// Mitsubishi GX Works2 project: 機電整合丙級第一題-ST   PLC: FX3U/FX3UC

// task Task_01 (event TRUE, interval 0, priority 31): POU_01

PROGRAM POU_01
VAR
  wProgramStep : INT;
  bM17 : BOOL;
  bM24 : BOOL;
  bM44 : BOOL;
  bM122 : BOOL;
  tdT22 : TON;
  bShape : BOOL;
  tdT24 : TON;
  tdT27 : TON;
  tdT29 : TON;
  bPB2 : BOOL;
  tdT123 : TON;
END_VAR
(* 機電整合丙級術科第一題
   Author: Steven Luo
   Date: 2018/09/26
*)

IF M8002 OR NOT X17 THEN (* 開機後或任何狀態按下急停 *)
	wProgramStep := 0;
	ZRST(TRUE, Y0, Y17);
	bM17 := FALSE;
	bM122 := FALSE;
END_IF;

IF NOT X17 THEN (* 按下急停 *)
	RST(TRUE, Y0);
	bM17 := TRUE;
END_IF;

IF X17 AND bM17 THEN (* 放開急停，等待復歸 *)
	wProgramStep := 122;
END_IF;

IF M8002 THEN
	wProgramStep := 21;
END_IF;

IF bM122 THEN
	IF M8013 THEN
		SET(TRUE, Y16); (* 黃燈閃爍 *)
	ELSE
		RST(TRUE, Y16);
	END_IF;
ELSE
	RST(TRUE, Y16);
END_IF;

CASE wProgramStep OF
	21:
		IF X1 AND X4 THEN
			SET(TRUE, Y17); (* 待機，綠燈亮、紅燈滅 *)
			RST(TRUE, Y15);
			RST(TRUE, Y2);
			tdT22(IN := FALSE);
			tdT24(IN := FALSE);
			tdT27(IN := FALSE);
			tdT29(IN := FALSE);
			tdT123(IN := FALSE);
			bM122 := FALSE;
			bM24 := FALSE;
			bM44 := FALSE;
			bPB2 := FALSE;
		END_IF;
		IF X13 AND X17 THEN
			IF X14 THEN (* 指定功能 *)
				RST(TRUE, Y2);
				RST(TRUE, Y4);
				RST(TRUE, Y5);
				IF X7 THEN (* PB1 *)
					SET(TRUE, Y2);
				ELSIF X4 AND X10 THEN (* PB2 *)
					IF X0 THEN
						RST(TRUE, Y0);
					ELSE
						SET(TRUE, Y0);
					END_IF;
				ELSIF X11 AND NOT X6 THEN (* PB3 *)
					SET(TRUE, Y4);
				ELSIF X12 AND NOT X4 THEN (* PB4 *)
					SET(TRUE, Y5);
				END_IF;
			ELSE
				IF X16 THEN (* 工作模式、按下啟動鈕 *)
					SET(TRUE, Y15); (* 紅燈亮、綠燈滅 *)
					RST(TRUE, Y17);
					wProgramStep := 22;
				END_IF;
			END_IF;
		END_IF;
	22:
		SET(TRUE, Y2); (* 輸送帶運轉 *)
		tdT29(IN := TRUE, PT := T#10s); (* 計時十秒 *)
		IF tdT29.Q THEN
			wProgramStep := 21;
		END_IF;
		IF X2 THEN
			tdT29(IN := FALSE);
			tdT22(IN := TRUE, PT := T#1s); (* 有料，計時一秒 *)
			IF tdT22.Q THEN
				RST(TRUE, Y2);
				IF X3 THEN (* 圓料 *)
					bShape := 1;
				ELSE (* 方料 *)
					bShape := 0;
				END_IF;
				wProgramStep := 23;
			END_IF;
		END_IF;
	23:
		SET(X4, Y0); (* 垂直缸下降 *)
		IF X0 THEN
			wProgramStep := 24;
		END_IF;
	24:
		SET(X4, Y6); (* 氣壓夾爪閉合 *)
		tdT24(IN := X4, PT := T#1s); (* 計時一秒 *)
		IF tdT24.Q THEN
			RST(X4, Y0); (* 垂直缸上升 *)
			wProgramStep := 25;
		END_IF;
	25:
		SET(X1, Y4); (* 龍門手臂左移，加X1限制避免撞機 *)
		IF bShape THEN (* 圓料 *)
			IF X5 THEN (* 到達圓料排料位 *)
				RST(X5, Y4);
				wProgramStep := 27;
			END_IF;
		ELSE (* 方料 *)
			IF X6 THEN (* 到達方料排料位 *)
				RST(X6, Y4);
				wProgramStep := 277;
			END_IF;
		END_IF;
	27:
		RST(X5, Y6); (* 螺桿機械手臂停止在圓料排料位 *)
		SET(X5, Y7); (* 氣壓夾爪打開 *)
		tdT27(IN := X5, PT := T#1s); (* 計時一秒 *)
		IF tdT27.Q THEN
			RST(TRUE, Y7);
			wProgramStep := 28;
		END_IF;
	28:
		SET(X1, Y5); (* 龍門手臂右移，加X1限制避免撞機 *)
		IF X4 THEN
			RST(TRUE, Y5);
			wProgramStep := 29;
		END_IF;
	29:
		IF X15 THEN
			tdT22(IN := FALSE);
			tdT24(IN := FALSE);
			tdT27(IN := FALSE);
			wProgramStep := 22;
		ELSE
			wProgramStep := 21;
		END_IF;
	122:
		IF NOT X13 AND X16 THEN (* 復歸模式、按下復歸開關 *)
			bM122 := TRUE;
			bM17 := FALSE;
			wProgramStep := 123;
		END_IF;
	123:
		SET(TRUE, Y7); (* 氣壓夾爪打開 *)
		tdT123(IN := TRUE, PT := T#1s); (* 計時一秒 *)
		IF tdT123.Q THEN
			RST(TRUE, Y7);
			wProgramStep := 124;
		END_IF;
	124:
		SET(NOT X4, Y5); (* 螺桿機械手臂右移 *)
		IF X4 THEN (* 回機械圓點 *)
			RST(TRUE, Y5);
			wProgramStep := 21;
		END_IF;
	277:
		SET(X6, Y0); (* 螺桿機械手臂停止在方料排料位，垂直缸下降 *)
		IF X0 THEN
			RST(X6, Y6); (* 氣壓夾爪打開 *)
			SET(X6, Y7);
			tdT27(IN := X6, PT := T#1s); (* 計時一秒 *)
			IF tdT27.Q THEN
				RST(TRUE, Y7);
				wProgramStep := 278;
			END_IF;
		END_IF;
	278:
		RST(X6, Y0); (* 垂直缸上升 *)
		wProgramStep := 28;
	ELSE
	;
END_CASE;
END_PROGRAM
